// TIA Portal V20 export
TYPE "LAF_typeSetPlcTime"
// Set new PLC time
// stored: Access Published
   STRUCT
      newDateAndTime : Date_And_Time;   // New PLC date and time that will be applied
      daylightSavingTime : Bool;   // TRUE = daylight saving time (first hour), FALSE = standard time (second hour)
      apply : Bool;   // Command to apply new time in the PLC
   END_STRUCT;
END_TYPE
